FUNCTION_BLOCK PAC_TransferWorkpieceTo_PSStart EXTENDS PAC_MoveWorkpiece_Base
VAR_INPUT
END_VAR
VAR_OUTPUT
END_VAR
VAR
	// (EProcessVariables.LSC_ProductType = 4) AND (EProcessVariables.PAC_WPNumber < 3)
	m_compExpr120: ComparisonExpression(EProcessVariables.LSC_ProductType, EComparisonType.equals, EDataType.numeric, FALSE, 4, '', TRUE);
	m_compExpr122: ComparisonExpression(EProcessVariables.PAC_WPNumber, EComparisonType.less, EDataType.numeric, FALSE, 3, '', TRUE);
	m_precondition: BoolExpression(m_compExpr120, EBoolOperation.and_op, m_compExpr122);
	
	// EProcessVariables.PAC_WPAtStart = TRUE
	m_postcondition: ComparisonExpression(EProcessVariables.PAC_WPAtStart, EComparisonType.equals, EDataType.binary, TRUE, 0, '', TRUE);
	
	m_timer: TON;
END_VAR

SUPER^();

METHOD PROTECTED  AtTarget : BOOL
VAR_INPUT
END_VAR
AtTarget := FALSE;

m_timer(IN := TRUE, PT := T#2000MS);
IF m_timer.Q THEN
	m_timer(IN := FALSE);
	m_ptrPAC^.METH_IncreaseWPNumberAtPAC();
	AtTarget := TRUE;
END_IF
END_METHOD

METHOD PROTECTED EjectOperation : BOOL
VAR_INPUT
END_VAR
//m_ptrPAC^.METH_IncreaseWPNumberAtPAC();
EjectOperation := TRUE;
END_METHOD

METHOD FB_init : BOOL
VAR_INPUT
	bInitRetains : BOOL; // if TRUE, the retain variables are initialized (warm start / cold start)
	bInCopyCode : BOOL;  // if TRUE, the instance afterwards gets moved into the copy code (online change)
	
	i_ptrPAC: POINTER TO PicAlphaConveyor;
END_VAR
m_ptrPAC := i_ptrPAC;

m_id := EPrimitives.PAC_TransferWorkpieceTo_PSStart;
m_timeout := T#200S;

Precondition := m_precondition;
Postcondition := m_postcondition;
END_METHOD

END_FUNCTION_BLOCK

(* stored: Version 1.1.0.1, ProductVersion 3.1.4024.9
   POU PAC_TransferWorkpieceTo_PSStart: Id {c6d8b21a-67b8-4abc-aeb4-548ca5ca0efd}, SpecialFunc None
   Method AtTarget: Id {67de37d6-5e26-48f6-b1ba-745a69378f53}
   Method EjectOperation: Id {536247b6-e0fd-4fab-870c-69d6d9f45706}
   Method FB_init: Id {eeb23bb6-e6d8-4e5e-ba00-5183307aab35} *)
